PROGRAM MANIPULATOR
VAR
	_context : fbManipulatorContext;
END_VAR

//_context.Run();

END_PROGRAM

(* stored: Version 1.1.0.1, ProductVersion 3.1.4024.6
   POU MANIPULATOR: Id {6ce25c6a-30a3-0b87-105c-f62d3a322039}, SpecialFunc None *)
